{attribute 'linkalways'} 
{attribute 'no_explicit_call' := 'This FB is a CLASS and must be accessed using methods or properties'}
{attribute 'enable_dynamic_creation'}
FUNCTION_BLOCK Node_F_VN_SetAt_TcVnPoint2_DINT EXTENDS VisionNode
VAR
    aElement : _TcVnPoint2_DINT;
    ipContainer : _ITcVnContainer;
    nIndex : _ULINT(0);
    hrPrev : _HRESULT(S_OK);
    hresult : _HRESULT(S_OK);
END_VAR

METHOD PUBLIC  Clone : I_Node
VAR
	pNode : POINTER TO Node_F_VN_SetAt_TcVnPoint2_DINT;
END_VAR
pNode := __NEW(Node_F_VN_SetAt_TcVnPoint2_DINT);
Clone := pNode^;
END_METHOD

METHOD FB_init : BOOL
VAR_INPUT
	bInitRetains : BOOL; // if TRUE, the retain variables are initialized (warm start / cold start)
	bInCopyCode : BOOL;  // if TRUE, the instance afterwards gets moved into the copy code (online change)
END_VAR
AddInput('aElement', aElement);
AddInput('ipContainer', ipContainer);
AddInput('nIndex', nIndex);
AddInput('hrPrev', hrPrev);
AddOutput('ipContainer', ipContainer);
AddOutput('hresult',hresult);
END_METHOD

METHOD PROTECTED OnExecute : HRESULT
hresult.Value := F_VN_SetAt_TcVnPoint2_DINT(
    aElement := aElement.Value,
    ipContainer := ipContainer.Value,
    nIndex := nIndex.Value,
    hrPrev:= hrPrev.Value);
END_METHOD

METHOD PUBLIC PreExecutionCheck
VAR_INPUT
	Check : I_PreExecutionChecks;
END_VAR
Check.IsTrue(ipContainer.IsValid, 'ipContainer must be a valid container');
END_METHOD

END_FUNCTION_BLOCK

(* stored: Version 1.1.0.1, ProductVersion 3.1.4024.13
   POU Node_F_VN_SetAt_TcVnPoint2_DINT: Id {9bc449f3-b7ca-4684-ba19-fd0f23e58586}, SpecialFunc None
   Folder Constructor: Id {1ef37a3a-f417-47d5-909b-561503a59277}
   Method Clone: Id {461876fd-e776-4241-9648-7aa540429661}
   Method FB_init: Id {b49deb5e-abb2-4a4f-8ef0-e7d1176103bf}
   Method OnExecute: Id {cfff9d15-5217-4e38-a78e-86acb020f053}
   Method PreExecutionCheck: Id {d9020cac-0cee-44a4-8c27-f2e304502606} *)
